FUNCTION_BLOCK RunningToReadyUnifiedProgramTransition EXTENDS RunningToReadyProgramTransition
VAR_STAT
	//! <summary>Class name shared by all instances of this function block.</summary>
	{attribute 'OPC.UA.DA' := '0'}
	_ClassName : STRING := __POUNAME();
END_VAR

{attribute 'monitoring' := 'call'}
PROPERTY ClassName : REFERENCE TO STRING
GET
ClassName REF= _ClassName;
END_GET
END_PROPERTY

END_FUNCTION_BLOCK

(* stored: Version 1.1.0.1
   POU RunningToReadyUnifiedProgramTransition: Id {126a1a70-fef6-448d-967b-c0b36ee85f5b}, SpecialFunc None
   Property ClassName: Id {4b679f9c-0b9b-4edd-8c2b-9c533a7ba7ab}
   Get Get: Id {b84226fb-e441-42ef-b90e-70bee2b5319e} *)
